PROGRAM MAIN
VAR
END_VAR

Global.touchData[0,0].x := Global.controller.TrackPadTouch0X;
Global.touchData[0,0].y := Global.controller.TrackPadTouch0Y;
Global.touchData[1,0].x := Global.controller.TrackPadTouch1X;
Global.touchData[1,0].y := Global.controller.TrackPadTouch1Y;

END_PROGRAM

(* stored: Version 1.1.0.1, ProductVersion 3.1.4024.9
   POU MAIN: Id {b79a84db-812c-4b01-916b-d0325876c153}, SpecialFunc None *)
